{attribute 'qualified_only'}
VAR_GLOBAL
	
	rX : REAL;
	rY : REAL;
	rZ : REAL;
	
	bB : BOOL;
	
END_VAR

(* stored: Version 1.1.0.1, ProductVersion 3.1.4024.13
   GVL GVL: Id {1119571a-e946-4415-97f1-8645da92f972} *)
